// SIMATIC STEP 7 (V5.x) project ZXX01_15_HSystem_RED_IO
// CPU: CPU 417-4 H
// CPU: CPU 417-4 H(1)
// station: Hardware
// station: SIMATIC H-Station(1)
// station: _S7H_BUSSYSTEM_CT
// program: S7 Program(1)
// program: S7-Programm(4)

SYMBOL_TABLE
"RED_IN"	FB 450	FB 450
"RED_OUT"	FB 451	FB 451
"RED_DIAG"	FB 452	FB 452
"RED_INIT"	FC 450	FC 450
"CYCL_EXC"	OB 1	OB 1	// Cycle Execution
"RED_I/O_FLT1"	OB 70	OB 70	// Redundancy I/O Fault 1
"RED_FLT"	OB 72	OB 72	// Redundancy Fault
"CYCL_FLT"	OB 80	OB 80	// Cycle Time Fault
"PS_FLT"	OB 81	OB 81	// Power Supply Fault
"I/O_FLT1"	OB 82	OB 82	// I/O Point Fault 1
"I/O_FLT2"	OB 83	OB 83	// I/O Point Fault 2
"OBNL_FLT"	OB 85	OB 85	// OB Not Loaded Fault
"RACK_FLT"	OB 86	OB 86	// Loss of Rack Fault
"COMM_FLT"	OB 87	OB 87	// Communication Fault
"COMPLETE RESTART"	OB 100	OB 100	// Complete Restart
"COLD RESTART"	OB 102	OB 102	// Cold Restart
"PROG_ERR"	OB 121	OB 121	// Programming Error
"MOD_ERR"	OB 122	OB 122	// Module Access Error
"WAIT"	SFC 47	SFC 47	// Delay Execution of the User Program
END_SYMBOL_TABLE

// FB 450: know-how protected block, not included

// FB 451: know-how protected block, not included

// FB 452: know-how protected block, not included

// FC 450: know-how protected block, not included

DATA_BLOCK DB 4
AUTHOR : RED_IO
FAMILY : RED_IO
VERSION : 0.0
"RED_DIAG"
BEGIN
END_DATA_BLOCK

DATA_BLOCK DB 5
AUTHOR : RED_IO
FAMILY : RED_IO
VERSION : 0.0
"RED_DIAG"
BEGIN
END_DATA_BLOCK

DATA_BLOCK DB 6
AUTHOR : RED_IO
FAMILY : RED_IO
VERSION : 0.0
"RED_DIAG"
BEGIN
END_DATA_BLOCK

DATA_BLOCK DB 7
AUTHOR : RED_IO
FAMILY : RED_IO
VERSION : 0.0
"RED_DIAG"
BEGIN
END_DATA_BLOCK

DATA_BLOCK DB 10
AUTHOR : RED_IO
FAMILY : RED_IO
VERSION : 0.0
"RED_IN"
BEGIN
END_DATA_BLOCK

DATA_BLOCK DB 11
AUTHOR : RED_IO
FAMILY : RED_IO
VERSION : 0.0
"RED_OUT"
BEGIN
END_DATA_BLOCK

ORGANIZATION_BLOCK "CYCL_EXC"	// OB 1
VERSION : 0.1
VAR_TEMP
  OB1_EV_CLASS : BYTE ;	//Bits 0-3 = 1 (Coming event), Bits 4-7 = 1 (Event class 1)
  OB1_SCAN_1 : BYTE ;	//1 (Cold restart scan 1 of OB 1), 3 (Scan 2-n of OB 1)
  OB1_PRIORITY : BYTE ;	//1 (Priority of 1 is lowest)
  OB1_OB_NUMBR : BYTE ;	//1 (Organization block 1, OB1)
  OB1_RESERVED_1 : BYTE ;	//Reserved for system
  OB1_RESERVED_2 : BYTE ;	//Reserved for system
  OB1_PREV_CYCLE : INT ;	//Cycle time of previous OB1 scan (milliseconds)
  OB1_MIN_CYCLE : INT ;	//Minimum cycle time of OB1 (milliseconds)
  OB1_MAX_CYCLE : INT ;	//Maximum cycle time of OB1 (milliseconds)
  OB1_DATE_TIME : DATE_AND_TIME ;	//Date and time OB1 started
END_VAR
BEGIN
NETWORK
TITLE =
      CALL  "RED_IN" , DB 10 (
           DIW 0                    := MW 10,
           DIW 2                    := MW 12);	//Redundant IO: Inputs
      AN    I 0.0;	//Counter (Byte 0)  on
      JC    next;
      L     QB 0;
      L     1;
      +I;
      T     QB 0;
next: AN    I 1.0;	// Shift (Byte 1)   on
      JC    ende;
      L     0;
      L     QB 1;
      <>I;
      JC    ug0;
      L     1;
      JU    con1;
ug0:  NOP   0;
      SLW   1;
con1: T     QB 1;
      CALL  "WAIT" (
           WT                       := 30000);
ende: NOP   0;
      CALL  "RED_OUT" , DB 11 (
           DIW 0                    := MW 14,
           DIW 2                    := MW 16);	//Redundant IO - Outputs
      BE;
END_ORGANIZATION_BLOCK

ORGANIZATION_BLOCK "RED_I/O_FLT1"	// OB 70
TITLE = "Redundancy I/O Fault 1"
VERSION : 0.0
VAR_TEMP
  OB70_EV_CLASS : BYTE ;	//Event class 7, module inserted/removed (8/9)
  OB70_FLT_ID : BYTE ;	//Fault identifcation code
  OB70_PRIORITY : BYTE ;	//25 (2...26, Priority of 1 is lowest)
  OB70_OB_NUMBR : BYTE ;	//70 (Organization block 70, OB70)
  OB70_INFO_1 : WORD ;	//Info 1
  OB70_INFO_2 : WORD ;	//Info 2
  OB70_INFO_3 : WORD ;	//Info 3
  OB70_RESERVED_1 : WORD ;	//Reserved for system
  OB70_DATE_TIME : DATE_AND_TIME ;	//Date and time OB70 started
END_VAR
BEGIN
// (block stored without names or comments; labels and parameter names are numbered)
END_ORGANIZATION_BLOCK

ORGANIZATION_BLOCK "RED_FLT"	// OB 72
TITLE = "Redundancy Fault"
VERSION : 0.0
VAR_TEMP
  OB72_EV_CLASS : BYTE ;	//Event class 7, module inserted/removed (8/9)
  OB72_FLT_ID : BYTE ;	//Fault identifcation code
  OB72_PRIORITY : BYTE ;	//Priority of OB Execution
  OB72_OB_NUMBR : BYTE ;	//72 (Organization block 72, OB72)
  OB72_RESERVED_1 : WORD ;	//Reserved for system
  OB72_INFO_1 : WORD ;	//Info 1
  OB72_INFO_2 : WORD ;	//Info 2
  OB72_INFO_3 : WORD ;	//Info 3
  OB72_DATE_TIME : DATE_AND_TIME ;	//Date and time OB72 started
END_VAR
BEGIN
NETWORK
TITLE =
      CALL  "RED_INIT" (
           $1                       := P#M 4.0,
           $2                       := P#M 6.0);
      CALL  "RED_DIAG" , DB 7 (
           DIW 0                    := MW 36,
           DIW 2                    := MW 38);
END_ORGANIZATION_BLOCK

ORGANIZATION_BLOCK "CYCL_FLT"	// OB 80
TITLE = "Cycle Time Fault"
VERSION : 0.0
VAR_TEMP
  OB80_EV_CLASS : BYTE ;	//16#35, Event class 3, Entering event state, Internal fault event
  OB80_FLT_ID : BYTE ;	//16#XX, Fault identifcation code
  OB80_PRIORITY : BYTE ;	//Priority of OB Execution
  OB80_OB_NUMBR : BYTE ;	//80 (Organization block 80, OB80)
  OB80_RESERVED_1 : BYTE ;	//Reserved for system
  OB80_RESERVED_2 : BYTE ;	//Reserved for system
  OB80_ERROR_INFO : WORD ;	//Error information on event
  OB80_ERR_EV_CLASS : BYTE ;	//Class of event causing error
  OB80_ERR_EV_NUM : BYTE ;	//Number of event causing error
  OB80_OB_PRIORITY : BYTE ;	//Priority of OB causing error
  OB80_OB_NUM : BYTE ;	//Number of OB causing error
  OB80_DATE_TIME : DATE_AND_TIME ;	//Date and time OB80 started
END_VAR
BEGIN
// (block stored without names or comments; labels and parameter names are numbered)
END_ORGANIZATION_BLOCK

ORGANIZATION_BLOCK "PS_FLT"	// OB 81
TITLE = "Power Supply Fault"
VERSION : 0.0
VAR_TEMP
  OB81_EV_CLASS : BYTE ;	//16#39, Event class 3, Entering event state, Internal fault event
  OB81_FLT_ID : BYTE ;	//16#XX, Fault identifcation code
  OB81_PRIORITY : BYTE ;	//26/28 (Priority of 1 is lowest)
  OB81_OB_NUMBR : BYTE ;	//81 (Organization block 81, OB81)
  OB81_RESERVED_1 : BYTE ;	//Reserved for system
  OB81_RESERVED_2 : BYTE ;	//Reserved for system
  OB81_MDL_ADDR : INT ;	//Reserved for system
  OB81_RESERVED_3 : BYTE ;	//Reserved for system
  OB81_RESERVED_4 : BYTE ;	//Reserved for system
  OB81_RESERVED_5 : BYTE ;	//Reserved for system
  OB81_RESERVED_6 : BYTE ;	//Reserved for system
  OB81_DATE_TIME : DATE_AND_TIME ;	//Date and time OB81 started
END_VAR
BEGIN
// (block stored without names or comments; labels and parameter names are numbered)
END_ORGANIZATION_BLOCK

ORGANIZATION_BLOCK "I/O_FLT1"	// OB 82
TITLE = "I/O Point Fault"
VERSION : 0.0
VAR_TEMP
  OB82_EV_CLASS : BYTE ;	//16#39, Event class 3, Entering event state, Internal fault event
  OB82_FLT_ID : BYTE ;	//16#XX, Fault identifcation code
  OB82_PRIORITY : BYTE ;	//Priority of OB Execution
  OB82_OB_NUMBR : BYTE ;	//82 (Organization block 82, OB82)
  OB82_RESERVED_1 : BYTE ;	//Reserved for system
  OB82_IO_FLAG : BYTE ;	//Input (01010100), Output (01010101)
  OB82_MDL_ADDR : WORD ;	//Base address of module with fault
  OB82_MDL_DEFECT : BOOL ;	//Module defective
  OB82_INT_FAULT : BOOL ;	//Internal fault
  OB82_EXT_FAULT : BOOL ;	//External fault
  OB82_PNT_INFO : BOOL ;	//Point information
  OB82_EXT_VOLTAGE : BOOL ;	//External voltage low
  OB82_FLD_CONNCTR : BOOL ;	//Field wiring connector missing
  OB82_NO_CONFIG : BOOL ;	//Module has no configuration data
  OB82_CONFIG_ERR : BOOL ;	//Module has configuration error
  OB82_MDL_TYPE : BYTE ;	//Type of module
  OB82_SUB_NDL_ERR : BOOL ;	//Sub-Module is missing or has error
  OB82_COMM_FAULT : BOOL ;	//Communication fault
  OB82_MDL_STOP : BOOL ;	//Module is stopped
  OB82_WTCH_DOG_FLT : BOOL ;	//Watch dog timer stopped module
  OB82_INT_PS_FLT : BOOL ;	//Internal power supply fault
  OB82_PRIM_BATT_FLT : BOOL ;	//Primary battery is in fault
  OB82_BCKUP_BATT_FLT : BOOL ;	//Backup battery is in fault
  OB82_RESERVED_2 : BOOL ;	//Reserved for system
  OB82_RACK_FLT : BOOL ;	//Rack fault, only for bus interface module
  OB82_PROC_FLT : BOOL ;	//Processor fault
  OB82_EPROM_FLT : BOOL ;	//EPROM fault
  OB82_RAM_FLT : BOOL ;	//RAM fault
  OB82_ADU_FLT : BOOL ;	//ADU fault
  OB82_FUSE_FLT : BOOL ;	//Fuse fault
  OB82_HW_INTR_FLT : BOOL ;	//Hardware interupt input in fault
  OB82_RESERVED_3 : BOOL ;	//Reserved for system
  OB82_DATE_TIME : DATE_AND_TIME ;	//Date and time OB82 started
END_VAR
BEGIN
NETWORK
TITLE =
      CALL  "RED_DIAG" , DB 4 (
           DIW 0                    := MW 20,
           DIW 2                    := MW 22);
END_ORGANIZATION_BLOCK

ORGANIZATION_BLOCK "I/O_FLT2"	// OB 83
TITLE = "I/O Point Fault"
VERSION : 0.0
VAR_TEMP
  OB83_EV_CLASS : BYTE ;	//16#38/39, Event class 3, module inserted/removed (8/9)
  OB83_FLT_ID : BYTE ;	//16#XX, Fault identifcation code
  OB83_PRIORITY : BYTE ;	//Priority of OB Execution
  OB83_OB_NUMBR : BYTE ;	//83 (Organization block 83, OB83)
  OB83_RESERVED_1 : BYTE ;	//Reserved for system
  OB83_MDL_ID : BYTE ;	//Input module (01010100), Output module (01010101)
  OB83_MDL_ADDR : WORD ;	//Base address of module with point fault
  OB83_RACK_NUM : INT ;	//Number of rack that has module with point fault
  OB83_MDL_TYPE : WORD ;	//Module type with point fault
  OB83_DATE_TIME : DATE_AND_TIME ;	//Date and time OB83 started
END_VAR
BEGIN
NETWORK
TITLE =
      CALL  "RED_DIAG" , DB 5 (
           DIW 0                    := MW 24,
           DIW 2                    := MW 26);
END_ORGANIZATION_BLOCK

ORGANIZATION_BLOCK "OBNL_FLT"	// OB 85
TITLE = "Organization Block (OB) Not Loaded Fault"
VERSION : 0.0
VAR_TEMP
  OB85_EV_CLASS : BYTE ;	//16#35 Event class 3
  OB85_FLT_ID : BYTE ;	//16#XX, Fault identification code
  OB85_PRIORITY : BYTE ;	//Priority of OB Execution
  OB85_OB_NUMBR : BYTE ;	//85 (Organization block 85, OB85)
  OB85_RESERVED_1 : BYTE ;	//Reserved for system
  OB85_RESERVED_2 : BYTE ;	//Reserved for system
  OB85_RESERVED_3 : INT ;	//Reserved for system
  OB85_ERR_EV_CLASS : BYTE ;	//Class of event causing error
  OB85_ERR_EV_NUM : BYTE ;	//Number of event causing error
  OB85_OB_PRIOR : BYTE ;	//Priority of OB causing error
  OB85_OB_NUM : BYTE ;	//Number of OB causing error
  OB85_DATE_TIME : DATE_AND_TIME ;	//Date and time OB85 started
END_VAR
BEGIN
NETWORK
TITLE =
      CALL  "RED_DIAG" , DB 6 (
           DIW 0                    := MW 28,
           DIW 2                    := MW 30);
END_ORGANIZATION_BLOCK

ORGANIZATION_BLOCK "RACK_FLT"	// OB 86
TITLE = "Loss Of Rack Fault"
VERSION : 0.0
VAR_TEMP
  OB86_EV_CLASS : BYTE ;	//16#38/39 Event class 3
  OB86_FLT_ID : BYTE ;	//16#C1/C4/C5, Fault identification code
  OB86_PRIORITY : BYTE ;	//26/28 (Priority of 1 is lowest)
  OB86_OB_NUMBR : BYTE ;	//86 (Organization block 86, OB86)
  OB86_RESERVED_1 : BYTE ;	//Reserved for system
  OB86_RESERVED_2 : BYTE ;	//Reserved for system
  OB86_MDL_ADDR : WORD ;	//Depending on fault identification code
  OB86_RACKS_FLTD : ARRAY  [0 .. 31 ] OF BOOL ;	//Racks in fault
  OB86_DATE_TIME : DATE_AND_TIME ;	//Date and time OB86 started
END_VAR
BEGIN
// (block stored without names or comments; labels and parameter names are numbered)
END_ORGANIZATION_BLOCK

ORGANIZATION_BLOCK "COMM_FLT"	// OB 87
TITLE = "Communication Fault"
VERSION : 0.0
VAR_TEMP
  OB87_EV_CLASS : BYTE ;	//16#35 Event class 3
  OB87_FLT_ID : BYTE ;	//16#XX, Fault identifcation code
  OB87_PRIORITY : BYTE ;	//26 (Priority of 1 is lowest)
  OB87_OB_NUMBR : BYTE ;	//87 (Organization block 87, OB87)
  OB87_RESERVED_1 : BYTE ;	//Reserved for system
  OB87_RESERVED_2 : BYTE ;	//Reserved for system
  OB87_RESERVED_3 : WORD ;	//Reserved for system
  OB87_RESERVED_4 : DWORD ;	//Reserved for system
  OB87_DATE_TIME : DATE_AND_TIME ;	//Date and time OB87 started
END_VAR
BEGIN
// (block stored without names or comments; labels and parameter names are numbered)
END_ORGANIZATION_BLOCK

ORGANIZATION_BLOCK "COMPLETE RESTART"	// OB 100
TITLE = "Complete Restart"
VERSION : 0.1
VAR_TEMP
  OB100_EV_CLASS : BYTE ;	//16#13, Event class 1, Entering event state, Event logged in diagnostic buffer
  OB100_STRTUP : BYTE ;	//16#81/82/83/84 Method of startup
  OB100_PRIORITY : BYTE ;	//Priority of OB Execution
  OB100_OB_NUMBR : BYTE ;	//100 (Organization block 100, OB100)
  OB100_RESERVED_1 : BYTE ;	//Reserved for system
  OB100_RESERVED_2 : BYTE ;	//Reserved for system
  OB100_STOP : WORD ;	//Event that caused CPU to stop (16#4xxx)
  OB100_STRT_INFO : DWORD ;	//Information on how system started
  OB100_DATE_TIME : DATE_AND_TIME ;	//Date and time OB100 started
END_VAR
BEGIN
NETWORK
TITLE =
      CALL  "RED_INIT" (
           $1                       := P#M 0.0,
           $2                       := P#M 2.0);
END_ORGANIZATION_BLOCK

ORGANIZATION_BLOCK "COLD RESTART"	// OB 102
TITLE = "Cold Restart"
VERSION : 0.1
VAR_TEMP
  OB102_EV_CLASS : BYTE ;	//16#13, Event class 1, Entering event state, Event logged in diagnostic buffer
  OB102_STRTUP : BYTE ;	//16#85...8B Method of startup
  OB102_PRIORITY : BYTE ;	//Priority of OB Execution
  OB102_OB_NUMBR : BYTE ;	//102 (Organization block 102, OB102)
  OB102_RESERVED_1 : BYTE ;	//Reserved for system
  OB102_RESERVED_2 : BYTE ;	//Reserved for system
  OB102_STOP : WORD ;	//Event that caused CPU to stop (16#4xxx)
  OB102_STRT_INFO : DWORD ;	//Information on how system started
  OB102_DATE_TIME : DATE_AND_TIME ;	//Date and time OB102 started
END_VAR
BEGIN
NETWORK
TITLE =
      CALL  "RED_INIT" (
           $1                       := P#M 0.0,
           $2                       := P#M 2.0);
END_ORGANIZATION_BLOCK

ORGANIZATION_BLOCK "PROG_ERR"	// OB 121
TITLE = "Programming Error"
VERSION : 0.0
VAR_TEMP
  OB121_EV_CLASS : BYTE ;	//16#25, Event class 2, Entering event state, Internal fault event
  OB121_SW_FLT : BYTE ;	//16#XX Software programming fault
  OB121_PRIORITY : BYTE ;	//X = Priority of OB where fault occured (Priority of 1 is lowest)
  OB121_OB_NUMBR : BYTE ;	//121 (Organization block 121, OB121)
  OB121_BLK_TYPE : BYTE ;	//16#88/8A/8B/8C/8E Type of block fault occured in
  OB121_RESERVED_1 : BYTE ;	//Reserved for system
  OB121_FLT_REG : WORD ;	//16#XX Specific register that caused fault
  OB121_BLK_NUM : WORD ;	//Number of block that programming fault occured in
  OB121_PRG_ADDR : WORD ;	//Address in block where programming fault occured
  OB121_DATE_TIME : DATE_AND_TIME ;	//Date and time OB121 started
END_VAR
BEGIN
// (block stored without names or comments; labels and parameter names are numbered)
END_ORGANIZATION_BLOCK

ORGANIZATION_BLOCK "MOD_ERR"	// OB 122
TITLE = "Module Access Error"
VERSION : 0.0
VAR_TEMP
  OB122_EV_CLASS : BYTE ;	//16#29, Event class 2, Entering event state, Internal fault event
  OB122_SW_FLT : BYTE ;	//16#XX Software error code
  OB122_PRIORITY : BYTE ;	//X = Priority of OB where fault occured (Priority of 1 is lowest)
  OB122_OB_NUMBR : BYTE ;	//122 (Organization block 122, OB122)
  OB122_BLK_TYPE : BYTE ;	//16#88/8A/8C/8E Type of block fault occured in
  OB122_MEM_AREA : BYTE ;	//Memory area where access error occured
  OB122_MEM_ADDR : WORD ;	//Memory address where access error occured
  OB122_BLK_NUM : WORD ;	//Block number in which error occured
  OB122_PRG_ADDR : WORD ;	//Program address where error occured
  OB122_DATE_TIME : DATE_AND_TIME ;	//Date and time OB1 started
END_VAR
BEGIN
// (block stored without names or comments; labels and parameter names are numbered)
END_ORGANIZATION_BLOCK

SYMBOL_TABLE
"WAIT"	SFC 47	SFC 47	// Delay Execution of the User Program
END_SYMBOL_TABLE

ORGANIZATION_BLOCK OB 1
VERSION : 0.1
VAR_TEMP
  OB1_EV_CLASS : BYTE ;	//Bits 0-3 = 1 (Coming event), Bits 4-7 = 1 (Event class 1)
  OB1_SCAN_1 : BYTE ;	//1 (Cold restart scan 1 of OB 1), 3 (Scan 2-n of OB 1)
  OB1_PRIORITY : BYTE ;	//1 (Priority of 1 is lowest)
  OB1_OB_NUMBR : BYTE ;	//1 (Organization block 1, OB1)
  OB1_RESERVED_1 : BYTE ;	//Reserved for system
  OB1_RESERVED_2 : BYTE ;	//Reserved for system
  OB1_PREV_CYCLE : INT ;	//Cycle time of previous OB1 scan (milliseconds)
  OB1_MIN_CYCLE : INT ;	//Minimum cycle time of OB1 (milliseconds)
  OB1_MAX_CYCLE : INT ;	//Maximum cycle time of OB1 (milliseconds)
  OB1_DATE_TIME : DATE_AND_TIME ;	//Date and time OB1 started
END_VAR
BEGIN
NETWORK
TITLE =
      AN    I 0.0;	//Counter (Byte 0)  on
      JC    next;
      L     QB 0;
      L     1;
      +I;
      T     QB 0;
next: AN    I 1.0;	// Shift (Byte 1)   on
      JC    ende;
      L     0;
      L     QB 1;
      <>I;
      JC    ug0;
      L     1;
      JU    con1;
ug0:  NOP   0;
      SLW   1;
con1: T     QB 1;
      CALL  "WAIT" (
           WT                       := 30000);
ende: BE;
END_ORGANIZATION_BLOCK

ORGANIZATION_BLOCK OB 70
TITLE = "Redundancy I/O Fault 1"
VERSION : 0.0
VAR_TEMP
  OB70_EV_CLASS : BYTE ;	//Event class 7, module inserted/removed (8/9)
  OB70_FLT_ID : BYTE ;	//Fault identifcation code
  OB70_PRIORITY : BYTE ;	//25 (2...26, Priority of 1 is lowest)
  OB70_OB_NUMBR : BYTE ;	//70 (Organization block 70, OB70)
  OB70_INFO_1 : WORD ;	//Info 1
  OB70_INFO_2 : WORD ;	//Info 2
  OB70_INFO_3 : WORD ;	//Info 3
  OB70_RESERVED_1 : WORD ;	//Reserved for system
  OB70_DATE_TIME : DATE_AND_TIME ;	//Date and time OB70 started
END_VAR
BEGIN
// (block stored without names or comments; labels and parameter names are numbered)
END_ORGANIZATION_BLOCK

ORGANIZATION_BLOCK OB 72
TITLE = "Redundancy Fault"
VERSION : 0.0
VAR_TEMP
  OB72_EV_CLASS : BYTE ;	//Event class 7, module inserted/removed (8/9)
  OB72_FLT_ID : BYTE ;	//Fault identifcation code
  OB72_PRIORITY : BYTE ;	//25 (2...26, Priority of 1 is lowest)
  OB72_OB_NUMBR : BYTE ;	//72 (Organization block 72, OB72)
  OB72_INFO_1 : WORD ;	//Info 1
  OB72_INFO_2 : WORD ;	//Info 2
  OB72_INFO_3 : WORD ;	//Info 3
  OB72_RESERVED_1 : WORD ;	//Reserved for system
  OB72_DATE_TIME : DATE_AND_TIME ;	//Date and time OB72 started
END_VAR
BEGIN
// (block stored without names or comments; labels and parameter names are numbered)
END_ORGANIZATION_BLOCK

ORGANIZATION_BLOCK OB 80
TITLE = "Cycle Time Fault"
VERSION : 0.0
VAR_TEMP
  OB80_EV_CLASS : BYTE ;	//16#35, Event class 3, Entering event state, Internal fault event
  OB80_FLT_ID : BYTE ;	//16#XX, Fault identifcation code
  OB80_PRIORITY : BYTE ;	//26 (Priority of 1 is lowest)
  OB80_OB_NUMBR : BYTE ;	//80 (Organization block 80, OB80)
  OB80_RESERVED_1 : BYTE ;	//Reserved for system
  OB80_RESERVED_2 : BYTE ;	//Reserved for system
  OB80_ERROR_INFO : WORD ;	//Error information on event
  OB80_ERR_EV_CLASS : BYTE ;	//Class of event causing error
  OB80_ERR_EV_NUM : BYTE ;	//Number of event causing error
  OB80_OB_PRIORITY : BYTE ;	//Priority of OB causing error
  OB80_OB_NUM : BYTE ;	//Number of OB causing error
  OB80_DATE_TIME : DATE_AND_TIME ;	//Date and time OB80 started
END_VAR
BEGIN
// (block stored without names or comments; labels and parameter names are numbered)
END_ORGANIZATION_BLOCK

ORGANIZATION_BLOCK OB 81
TITLE = "Power Supply Fault"
VERSION : 0.0
VAR_TEMP
  OB81_EV_CLASS : BYTE ;	//16#39, Event class 3, Entering event state, Internal fault event
  OB81_FLT_ID : BYTE ;	//16#XX, Fault identifcation code
  OB81_PRIORITY : BYTE ;	//26/28 (Priority of 1 is lowest)
  OB81_OB_NUMBR : BYTE ;	//81 (Organization block 81, OB81)
  OB81_RESERVED_1 : BYTE ;	//Reserved for system
  OB81_RESERVED_2 : BYTE ;	//Reserved for system
  OB81_MDL_ADDR : INT ;	//Reserved for system
  OB81_RESERVED_3 : BYTE ;	//Reserved for system
  OB81_RESERVED_4 : BYTE ;	//Reserved for system
  OB81_RESERVED_5 : BYTE ;	//Reserved for system
  OB81_RESERVED_6 : BYTE ;	//Reserved for system
  OB81_DATE_TIME : DATE_AND_TIME ;	//Date and time OB81 started
END_VAR
BEGIN
// (block stored without names or comments; labels and parameter names are numbered)
END_ORGANIZATION_BLOCK

ORGANIZATION_BLOCK OB 82
TITLE = "I/O Point Fault"
VERSION : 0.0
VAR_TEMP
  OB82_EV_CLASS : BYTE ;	//16#39, Event class 3, Entering event state, Internal fault event
  OB82_FLT_ID : BYTE ;	//16#XX, Fault identifcation code
  OB82_PRIORITY : BYTE ;	//26/28 (Priority of 1 is lowest)
  OB82_OB_NUMBR : BYTE ;	//82 (Organization block 82, OB82)
  OB82_RESERVED_1 : BYTE ;	//Reserved for system
  OB82_IO_FLAG : BYTE ;	//Input (01010100), Output (01010101)
  OB82_MDL_ADDR : INT ;	//Base address of module with fault
  OB82_MDL_DEFECT : BOOL ;	//Module defective
  OB82_INT_FAULT : BOOL ;	//Internal fault
  OB82_EXT_FAULT : BOOL ;	//External fault
  OB82_PNT_INFO : BOOL ;	//Point information
  OB82_EXT_VOLTAGE : BOOL ;	//External voltage low
  OB82_FLD_CONNCTR : BOOL ;	//Field wiring connector missing
  OB82_NO_CONFIG : BOOL ;	//Module has no configuration data
  OB82_CONFIG_ERR : BOOL ;	//Module has configuration error
  OB82_MDL_TYPE : BYTE ;	//Type of module
  OB82_SUB_NDL_ERR : BOOL ;	//Sub-Module is missing or has error
  OB82_COMM_FAULT : BOOL ;	//Communication fault
  OB82_MDL_STOP : BOOL ;	//Module is stopped
  OB82_WTCH_DOG_FLT : BOOL ;	//Watch dog timer stopped module
  OB82_INT_PS_FLT : BOOL ;	//Internal power supply fault
  OB82_PRIM_BATT_FLT : BOOL ;	//Primary battery is in fault
  OB82_BCKUP_BATT_FLT : BOOL ;	//Backup battery is in fault
  OB82_RESERVED_2 : BOOL ;	//Reserved for system
  OB82_RACK_FLT : BOOL ;	//Rack fault, only for bus interface module
  OB82_PROC_FLT : BOOL ;	//Processor fault
  OB82_EPROM_FLT : BOOL ;	//EPROM fault
  OB82_RAM_FLT : BOOL ;	//RAM fault
  OB82_ADU_FLT : BOOL ;	//ADU fault
  OB82_FUSE_FLT : BOOL ;	//Fuse fault
  OB82_HW_INTR_FLT : BOOL ;	//Hardware interupt input in fault
  OB82_RESERVED_3 : BOOL ;	//Reserved for system
  OB82_DATE_TIME : DATE_AND_TIME ;	//Date and time OB82 started
END_VAR
BEGIN
// (block stored without names or comments; labels and parameter names are numbered)
END_ORGANIZATION_BLOCK

ORGANIZATION_BLOCK OB 83
TITLE = "I/O Point Fault"
VERSION : 0.0
VAR_TEMP
  OB83_EV_CLASS : BYTE ;	//16#38/39, Event class 3, module inserted/removed (8/9)
  OB83_FLT_ID : BYTE ;	//16#XX, Fault identifcation code
  OB83_PRIORITY : BYTE ;	//26/28 (Priority of 1 is lowest)
  OB83_OB_NUMBR : BYTE ;	//83 (Organization block 83, OB83)
  OB83_RESERVED_1 : BYTE ;	//Reserved for system
  OB83_MDL_ID : BYTE ;	//Input module (01010100), Output module (01010101)
  OB83_MDL_ADDR : WORD ;	//Base address of module with point fault
  OB83_RACK_NUM : WORD ;	//Number of rack that has module with point fault
  OB83_MDL_TYPE : WORD ;	//Module type with point fault
  OB83_DATE_TIME : DATE_AND_TIME ;	//Date and time OB83 started
END_VAR
BEGIN
// (block stored without names or comments; labels and parameter names are numbered)
END_ORGANIZATION_BLOCK

ORGANIZATION_BLOCK OB 85
TITLE = "Organization Block (OB) Not Loaded Fault"
VERSION : 0.0
VAR_TEMP
  OB85_EV_CLASS : BYTE ;	//16#35 Event class 3
  OB85_FLT_ID : BYTE ;	//16#XX, Fault identification code
  OB85_PRIORITY : BYTE ;	//26 (Priority of 1 is lowest)
  OB85_OB_NUMBR : BYTE ;	//85 (Organization block 85, OB85)
  OB85_RESERVED_1 : BYTE ;	//Reserved for system
  OB85_RESERVED_2 : BYTE ;	//Reserved for system
  OB85_RESERVED_3 : INT ;	//Reserved for system
  OB85_ERR_EV_CLASS : BYTE ;	//Class of event causing error
  OB85_ERR_EV_NUM : BYTE ;	//Number of event causing error
  OB85_OB_PRIOR : BYTE ;	//Priority of OB causing error
  OB85_OB_NUM : BYTE ;	//Number of OB causing error
  OB85_DATE_TIME : DATE_AND_TIME ;	//Date and time OB85 started
END_VAR
BEGIN
// (block stored without names or comments; labels and parameter names are numbered)
END_ORGANIZATION_BLOCK

ORGANIZATION_BLOCK OB 86
TITLE = "Loss Of Rack Fault"
VERSION : 0.0
VAR_TEMP
  OB86_EV_CLASS : BYTE ;	//16#38/39 Event class 3
  OB86_FLT_ID : BYTE ;	//16#C1/C4/C5, Fault identification code
  OB86_PRIORITY : BYTE ;	//26/28 (Priority of 1 is lowest)
  OB86_OB_NUMBR : BYTE ;	//86 (Organization block 86, OB86)
  OB86_RESERVED_1 : BYTE ;	//Reserved for system
  OB86_RESERVED_2 : BYTE ;	//Reserved for system
  OB86_MDL_ADDR : WORD ;	//Depending on fault identification code
  OB86_RACKS_FLTD : ARRAY  [0 .. 31 ] OF BOOL ;	//Racks in fault
  OB86_DATE_TIME : DATE_AND_TIME ;	//Date and time OB86 started
END_VAR
BEGIN
// (block stored without names or comments; labels and parameter names are numbered)
END_ORGANIZATION_BLOCK

ORGANIZATION_BLOCK OB 87
TITLE = "Communication Fault"
VERSION : 0.0
VAR_TEMP
  OB87_EV_CLASS : BYTE ;	//16#35 Event class 3
  OB87_FLT_ID : BYTE ;	//16#XX, Fault identifcation code
  OB87_PRIORITY : BYTE ;	//26 (Priority of 1 is lowest)
  OB87_OB_NUMBR : BYTE ;	//87 (Organization block 87, OB87)
  OB87_RESERVED_1 : BYTE ;	//Reserved for system
  OB87_RESERVED_2 : BYTE ;	//Reserved for system
  OB87_RESERVED_3 : WORD ;	//Reserved for system
  OB87_RESERVED_4 : DWORD ;	//Reserved for system
  OB87_DATE_TIME : DATE_AND_TIME ;	//Date and time OB87 started
END_VAR
BEGIN
// (block stored without names or comments; labels and parameter names are numbered)
END_ORGANIZATION_BLOCK

ORGANIZATION_BLOCK OB 121
TITLE = "Programming Error"
VERSION : 0.0
VAR_TEMP
  OB121_EV_CLASS : BYTE ;	//16#25, Event class 2, Entering event state, Internal fault event
  OB121_SW_FLT : BYTE ;	//16#XX Software programming fault
  OB121_PRIORITY : BYTE ;	//X = Priority of OB where fault occured (Priority of 1 is lowest)
  OB121_OB_NUMBR : BYTE ;	//121 (Organization block 121, OB121)
  OB121_BLK_TYPE : BYTE ;	//16#88/8A/8B/8C/8E Type of block fault occured in
  OB121_RESERVED_1 : BYTE ;	//Reserved for system
  OB121_FLT_REG : WORD ;	//16#XX Specific register that caused fault
  OB121_BLK_NUM : WORD ;	//Number of block that programming fault occured in
  OB121_PRG_ADDR : WORD ;	//Address in block where programming fault occured
  OB121_DATE_TIME : DATE_AND_TIME ;	//Date and time OB121 started
END_VAR
BEGIN
// (block stored without names or comments; labels and parameter names are numbered)
END_ORGANIZATION_BLOCK

ORGANIZATION_BLOCK OB 122
TITLE = "Module Access Error"
VERSION : 0.0
VAR_TEMP
  OB122_EV_CLASS : BYTE ;	//16#29, Event class 2, Entering event state, Internal fault event
  OB122_SW_FLT : BYTE ;	//16#XX Software error code
  OB122_PRIORITY : BYTE ;	//X = Priority of OB where fault occured (Priority of 1 is lowest)
  OB122_OB_NUMBR : BYTE ;	//122 (Organization block 122, OB122)
  OB122_BLK_TYPE : BYTE ;	//16#88/8A/8C/8E Type of block fault occured in
  OB122_MEM_AREA : BYTE ;	//Memory area where access error occured
  OB122_MEM_ADDR : WORD ;	//Memory address where access error occured
  OB122_BLK_NUM : WORD ;	//Block number in which error occured
  OB122_PRG_ADDR : WORD ;	//Program address where error occured
  OB122_DATE_TIME : DATE_AND_TIME ;	//Date and time OB1 started
END_VAR
BEGIN
// (block stored without names or comments; labels and parameter names are numbered)
END_ORGANIZATION_BLOCK
